# EPICS autosave request: softGlueApp/Db/Shift_settings.req
$(P)$(H)Shift-$(N)_desc
$(P)$(H)Shift-$(N)_LOADVAL
$(P)$(H)Shift-$(N)_D_Signal
$(P)$(H)Shift-$(N)_CLOCK_Signal
$(P)$(H)Shift-$(N)_LOAD_Signal
$(P)$(H)Shift-$(N)_Q_Signal
